TYPE
    SyncUnitsBase_AD6C35CE :
    STRUCT
    END_STRUCT
END_TYPE

(* stored: Version 1.1.0.1, ProductVersion 3.1.4024.12
   DUT SyncUnitsBase_AD6C35CE: Id {77296da9-7498-0b40-1926-b8a7ed67137d} *)
